{attribute addProperty BoxType "EL6201-0000-0017"}
{attribute addProperty Id "Slave_26A_DO0BIT10.125201Slave_26A_DO1BIT10.125202Slave_26A_DO2BIT10.125203Slave_26A_DO3BIT10.125204Slave_26B_DO0BIT10.125205Slave_26B_DO1BIT10.125206Slave_26B_DO2BIT10.125207Slave_26B_DO3BIT10.125208"}
{attribute addProperty CRC "2378885056"}
{attribute addProperty SizeInBites "8"}
{attribute addProperty SizeInBytes "1"}
TYPE Slave_26_Outputs_8DCAE7C0 :
STRUCT
	{attribute addProperty Name "Slave_26A_DO0"}
	Slave_26A_DO0 : BIT;
	{attribute addProperty Name "Slave_26A_DO1"}
	Slave_26A_DO1 : BIT;
	{attribute addProperty Name "Slave_26A_DO2"}
	Slave_26A_DO2 : BIT;
	{attribute addProperty Name "Slave_26A_DO3"}
	Slave_26A_DO3 : BIT;
	{attribute addProperty Name "Slave_26B_DO0"}
	Slave_26B_DO0 : BIT;
	{attribute addProperty Name "Slave_26B_DO1"}
	Slave_26B_DO1 : BIT;
	{attribute addProperty Name "Slave_26B_DO2"}
	Slave_26B_DO2 : BIT;
	{attribute addProperty Name "Slave_26B_DO3"}
	Slave_26B_DO3 : BIT;
END_STRUCT
END_TYPE

(* stored: Version 1.2.0.0, ProductVersion 3.1.4024.9
   DUT Slave_26_Outputs_8DCAE7C0: Id {ac4a863e-d979-4aef-bc22-73af8cf00d52} *)
